PROGRAM LaserMarking_Variable_Selection
VAR
END_VAR

END_PROGRAM

(* stored: Version 1.1.0.1, ProductVersion 3.1.4024.0
   POU LaserMarking_Variable_Selection: Id {f494b5d2-9612-49b8-a0ce-4177ac483716}, SpecialFunc None *)
